(* PLC project Beremiz Supervised Raw Ethernet Study PLC, Study Stand Beremiz Supervised Raw PLC 1 *)
(* stored: creationDateTime 2026-06-15T12:00:00, modificationDateTime 2026-06-15T12:00:00 *)

PROGRAM plc_prg
  VAR_EXTERNAL
    RawSensorValue : UINT;
    RawThreshold : UINT;
    RawForcedOutput : UINT;
    RawSequence : UDINT;
    RawOutputCommand : UINT;
  END_VAR
  VAR
    sensor_value : UINT;
    threshold : UINT;
    remote_output_echo : UINT;
    sequence : UDINT;
    alarm : BOOL;
    output_command : UINT;
    request_count : UDINT;
    high_request_count : UDINT;
    low_request_count : UDINT;
    last_sequence : UDINT;
    sequence_changed : BOOL;
    request_seen : BOOL;
  END_VAR

            sensor_value := RawSensorValue;
threshold := RawThreshold;
remote_output_echo := RawForcedOutput;
sequence := RawSequence;

alarm := sensor_value > threshold;

sequence_changed := (NOT request_seen) OR (sequence <> last_sequence);

IF sequence_changed THEN
    request_count := request_count + UDINT#1;

    IF alarm THEN
        high_request_count := high_request_count + UDINT#1;
    ELSE
        low_request_count := low_request_count + UDINT#1;
    END_IF;

    last_sequence := sequence;
    request_seen := TRUE;
END_IF;

IF alarm THEN
    output_command := UINT#1;
ELSE
    output_command := UINT#0;
END_IF;

RawOutputCommand := output_command;
          
END_PROGRAM

CONFIGURATION config
  RESOURCE resource1 ON PLC
    TASK task0(INTERVAL := T#1ms, PRIORITY := 0);
    PROGRAM instance0 WITH task0 : plc_prg;
  END_RESOURCE
END_CONFIGURATION
